// Mitsubishi GX Works2 project: PLC_GROUP6   PLC: FX3G

// global labels: Global1
VAR_GLOBAL
  startDay AT X007 : BOOL;
  lifeDay AT Y007 : BOOL;
  stayOn AT Y007 : BOOL;
  Dgima AT X001 : BOOL;
  AnalogInput1 AT D8280 : INT;
  beerType AT D1502 : REAL;
END_VAR
VAR_GLOBAL CONSTANT
  SHMARIMfor6_lagger : REAL := 150;
  LETETfor6_lagger : REAL := 12;
  KSHUTfor6_lagger : REAL := 60;
  SHMARIMfor6_pilzner : REAL := 120;
  LETETfor6_pilzner : REAL := 6;
  KSHUTfor6_pilzner : REAL := 54;
END_VAR
VAR_GLOBAL
  timerForCooking AT TC1 : BOOL;
END_VAR
VAR_GLOBAL CONSTANT
  secondsCooking : INT := 40;
END_VAR
VAR_GLOBAL
  EndCooking AT TS1 : BOOL;
  cooking AT Y001 : BOOL;
  stopCooking AT Y001 : BOOL;
  startTsisa AT X005 : BOOL;
  M0helper AT M0 : BOOL;
END_VAR
VAR_GLOBAL CONSTANT
  OnOf : INT := 5;
END_VAR
VAR_GLOBAL
  OnOfTsisa AT TC2 : BOOL;
  firstBulb AT TS2 : BOOL;
  first AT Y003 : BOOL;
  OnOfTsisa2 AT TC3 : BOOL;
  secondBulb AT TS3 : BOOL;
  second AT Y004 : BOOL;
  stopTsisa1 AT Y003 : BOOL;
  stopTsisa2 AT Y004 : BOOL;
  startAriza AT X002 : BOOL;
  arizat1Bottle AT X000 : BOOL;
  startMore5 AT Y002 : BOOL;
  countBottles AT CC1 : BOOL;
END_VAR
VAR_GLOBAL CONSTANT
  counterBottles : INT := 6;
END_VAR
VAR_GLOBAL
  finishCount AT CS1 : BOOL;
  endDay AT X011 : BOOL;
END_VAR
VAR_GLOBAL CONSTANT
  counterFirstBottle : INT := 1;
END_VAR
VAR_GLOBAL
  countFirstBottle AT CC0 : BOOL;
  startCount AT CS0 : BOOL;
  AddSixBeer AT Y002 : BOOL;
END_VAR
VAR_GLOBAL CONSTANT
  AddingSixBeer : REAL := 1.0;
END_VAR
VAR_GLOBAL
  validAmount AT M2 : BOOL;
  shmarim_Input AT D1100 : REAL;
  letet_Input AT D1200 : REAL;
  kshut_Input AT D1300 : REAL;
END_VAR
VAR_GLOBAL CONSTANT
  Min_shmarim : REAL := 120.0;
  Min_letet : REAL := 6.0;
  Min_kshut : REAL := 54.0;
END_VAR
VAR_GLOBAL
  shmarim_TOT AT D1102 : REAL;
  letet_TOT AT D1202 : REAL;
  kshut_TOT AT D1302 : REAL;
END_VAR
VAR_GLOBAL CONSTANT
  MinPIZ : REAL := 6.0;
END_VAR
VAR_GLOBAL
  checkValid AT M1 : BOOL;
  AmountSixBeer AT D1402 : REAL;
END_VAR
VAR_GLOBAL CONSTANT
  Normaliz : REAL := 404.5;
  MinLAG : REAL;
  MAXLAG : REAL := 5.0;
END_VAR
VAR_GLOBAL
  LAGChoose AT M3 : BOOL;
  PIZChoose AT M4 : BOOL;
  tsisaOfPIZ AT TC14 : BOOL;
  tsisaOfLAG AT TC13 : BOOL;
END_VAR
VAR_GLOBAL CONSTANT
  tsisaLAG : INT := 30;
  tsisaPIZ : INT := 40;
END_VAR
VAR_GLOBAL
  finishTSISAlag AT TS13 : BOOL;
  finishTSISApiz AT TS14 : BOOL;
  endOneIteration AT M10 : BOOL;
  theDayEnd AT M20 : BOOL;
END_VAR
VAR_GLOBAL CONSTANT
  constant_40 : REAL := 40;
END_VAR
VAR_GLOBAL
  Output_SixBeer AT D1404 : REAL;
  analogOutput AT D8282 : INT;
  checkMLAY AT M13 : BOOL;
END_VAR
VAR_GLOBAL CONSTANT
  bishul6LAG : REAL := 222;
END_VAR
VAR_GLOBAL
  bishul_TOT AT D1600 : REAL;
END_VAR
VAR_GLOBAL CONSTANT
  bishul6pilzner : REAL := 180;
END_VAR
VAR_GLOBAL
  tsisa_TOT AT D1602 : REAL;
  helpDayOn AT M22 : BOOL;
  endDayFINISH AT M11 : BOOL;
  MlayEndDay AT M12 : BOOL;
END_VAR

// task Task_01 (event TRUE, interval 0, priority 31): POU_01

PROGRAM POU_01
(* structured ladder/FBD written out as ST: instructions are called as NAME(EN, inputs, outputs); _pN, _eN, _tN stand for wires *)
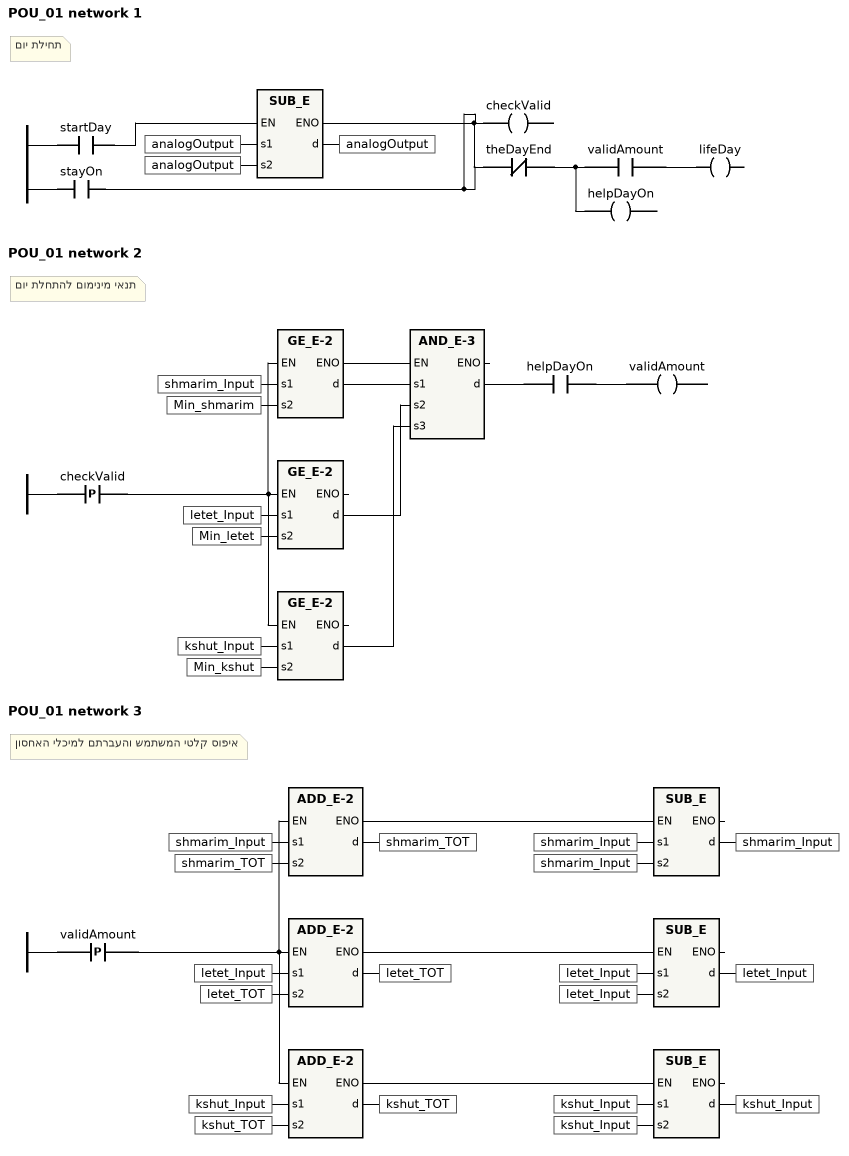
(* network 1 *)
(* תחילת יום *)
_e1 := SUB_E(startDay, analogOutput, analogOutput, analogOutput);
_p2 := _e1 OR stayOn;
checkValid := _p2;
_p3 := _p2 AND NOT theDayEnd;
lifeDay := _p3 AND validAmount;
helpDayOn := _p3;
(* network 2 *)
(* תנאי מינימום להתחלת יום *)
_p1 := LDP(TRUE, checkValid);
_e3 := GE_E(_p1, shmarim_Input, Min_shmarim, _t2);
GE_E(_p1, letet_Input, Min_letet, _t4);
GE_E(_p1, kshut_Input, Min_kshut, _t5);
AND_E(_e3, _t2, _t4, _t5, _t6);
validAmount := _t6 AND helpDayOn;
(* network 3 *)
(* איפוס קלטי המשתמש והעברתם למיכלי האחסון *)
_p1 := LDP(TRUE, validAmount);
_e2 := ADD_E(_p1, shmarim_Input, shmarim_TOT, shmarim_TOT);
SUB_E(_e2, shmarim_Input, shmarim_Input, shmarim_Input);
_e3 := ADD_E(_p1, letet_Input, letet_TOT, letet_TOT);
SUB_E(_e3, letet_Input, letet_Input, letet_Input);
_e4 := ADD_E(_p1, kshut_Input, kshut_TOT, kshut_TOT);
SUB_E(_e4, kshut_Input, kshut_Input, kshut_Input);
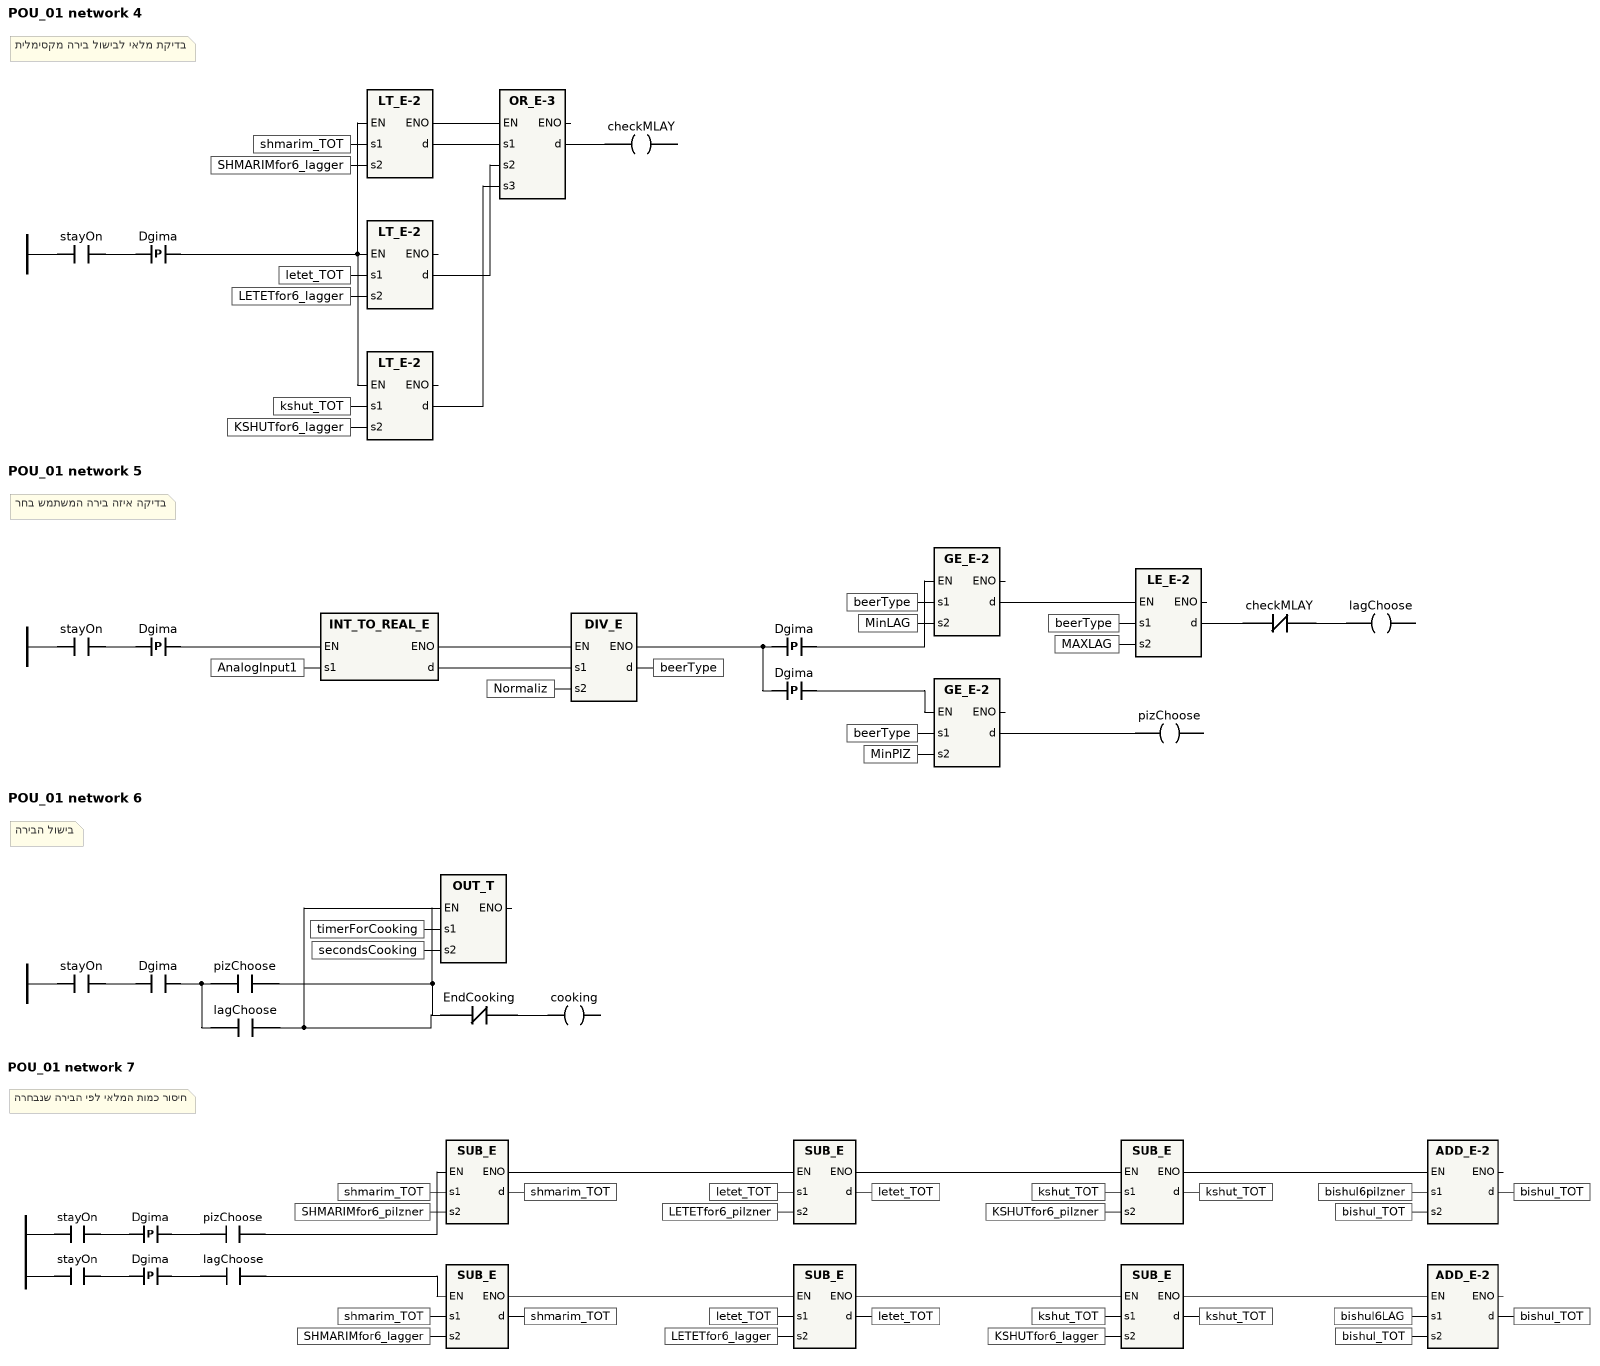
(* network 4 *)
(* בדיקת מלאי לבישול בירה מקסימלית *)
_p1 := stayOn AND LDP(TRUE, Dgima);
_e3 := LT_E(_p1, shmarim_TOT, SHMARIMfor6_lagger, _t2);
LT_E(_p1, letet_TOT, LETETfor6_lagger, _t4);
LT_E(_p1, kshut_TOT, KSHUTfor6_lagger, _t5);
OR_E(_e3, _t2, _t4, _t5, _t6);
checkMLAY := _t6;
(* network 5 *)
(* בדיקה איזה בירה המשתמש בחר *)
_e2 := INT_TO_REAL_E(stayOn AND LDP(TRUE, Dgima), AnalogInput1, _t1);
_e3 := DIV_E(_e2, _t1, Normaliz, beerType);
GE_E(_e3 AND LDP(TRUE, Dgima), beerType, MinLAG, _t4);
LE_E(_t4, beerType, MAXLAG, _t5);
lagChoose := _t5 AND NOT checkMLAY;
GE_E(_e3 AND LDP(TRUE, Dgima), beerType, MinPIZ, _t6);
pizChoose := _t6;
(* network 6 *)
(* בישול הבירה *)
_p1 := stayOn AND Dgima;
_p2 := (_p1 AND pizChoose) OR (_p1 AND lagChoose);
OUT_T(_p2, timerForCooking, secondsCooking);
cooking := _p2 AND NOT EndCooking;
(* network 7 *)
(* חיסור כמות המלאי לפי הבירה שנבחרה *)
_e1 := SUB_E(stayOn AND LDP(TRUE, Dgima) AND pizChoose, shmarim_TOT, SHMARIMfor6_pilzner, shmarim_TOT);
_e2 := SUB_E(_e1, letet_TOT, LETETfor6_pilzner, letet_TOT);
_e3 := SUB_E(_e2, kshut_TOT, KSHUTfor6_pilzner, kshut_TOT);
ADD_E(_e3, bishul6pilzner, bishul_TOT, bishul_TOT);
_e4 := SUB_E(stayOn AND LDP(TRUE, Dgima) AND lagChoose, shmarim_TOT, SHMARIMfor6_lagger, shmarim_TOT);
_e5 := SUB_E(_e4, letet_TOT, LETETfor6_lagger, letet_TOT);
_e6 := SUB_E(_e5, kshut_TOT, KSHUTfor6_lagger, kshut_TOT);
ADD_E(_e6, bishul6LAG, bishul_TOT, bishul_TOT);
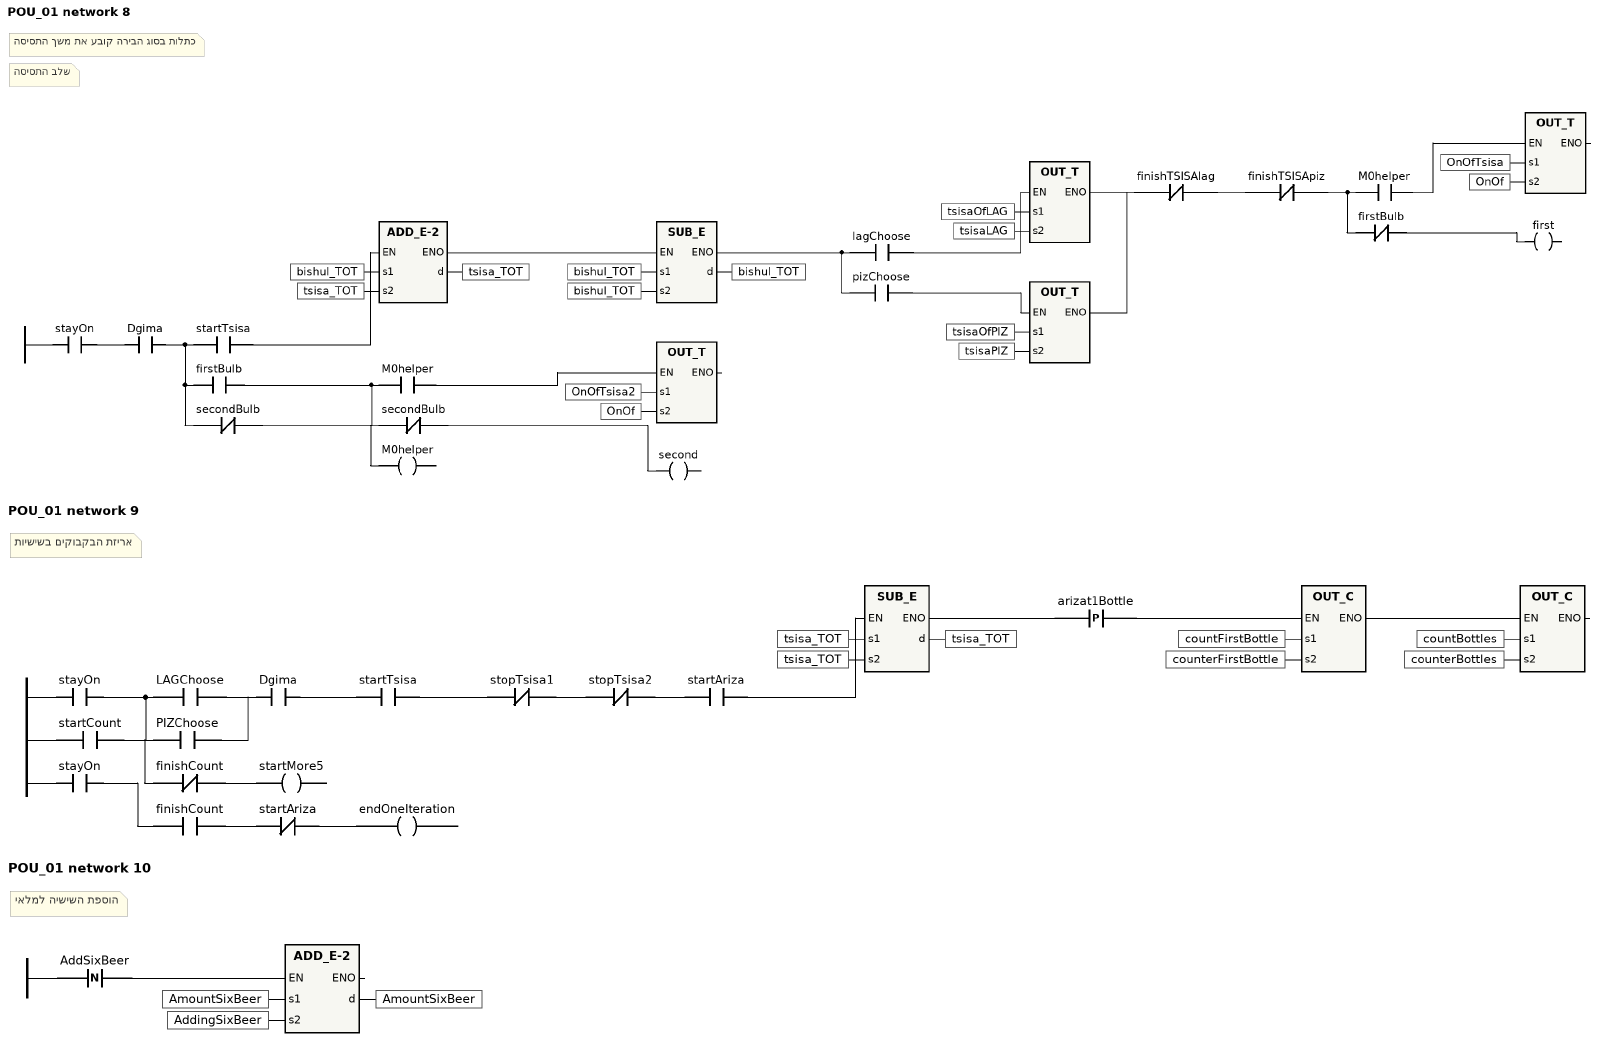
(* network 8 *)
(* כתלות בסוג הבירה קובע את משך התסיסה *)
(* שלב התסיסה *)
_p1 := stayOn AND Dgima;
_e2 := ADD_E(_p1 AND startTsisa, bishul_TOT, tsisa_TOT, tsisa_TOT);
_e3 := SUB_E(_e2, bishul_TOT, bishul_TOT, bishul_TOT);
_e4 := OUT_T(_e3 AND lagChoose, tsisaOfLAG, tsisaLAG);
_e5 := OUT_T(_e3 AND pizChoose, tsisaOfPIZ, tsisaPIZ);
_p6 := ((_e4 OR _e5) AND NOT finishTSISAlag) AND NOT finishTSISApiz;
OUT_T(_p6 AND M0helper, OnOfTsisa, OnOf);
first := _p6 AND NOT firstBulb;
_p7 := _p1 AND firstBulb;
OUT_T(_p7 AND M0helper, OnOfTsisa2, OnOf);
second := _p7 AND NOT secondBulb;
M0helper := _p1 AND NOT secondBulb;
(* network 9 *)
(* אריזת הבקבוקים בשישיות *)
_e1 := SUB_E(((((((stayOn AND LAGChoose) OR (stayOn AND PIZChoose)) AND Dgima) AND startTsisa) AND NOT stopTsisa1) AND NOT stopTsisa2) AND startAriza, tsisa_TOT, tsisa_TOT, tsisa_TOT);
_e2 := OUT_C(_e1 AND LDP(TRUE, arizat1Bottle), countFirstBottle, counterFirstBottle);
OUT_C(_e2, countBottles, counterBottles);
startMore5 := startCount AND NOT finishCount;
endOneIteration := stayOn AND finishCount AND NOT startAriza;
(* network 10 *)
(* הוספת השישיה למלאי *)
ADD_E(LDF(TRUE, AddSixBeer), AmountSixBeer, AddingSixBeer, AmountSixBeer);
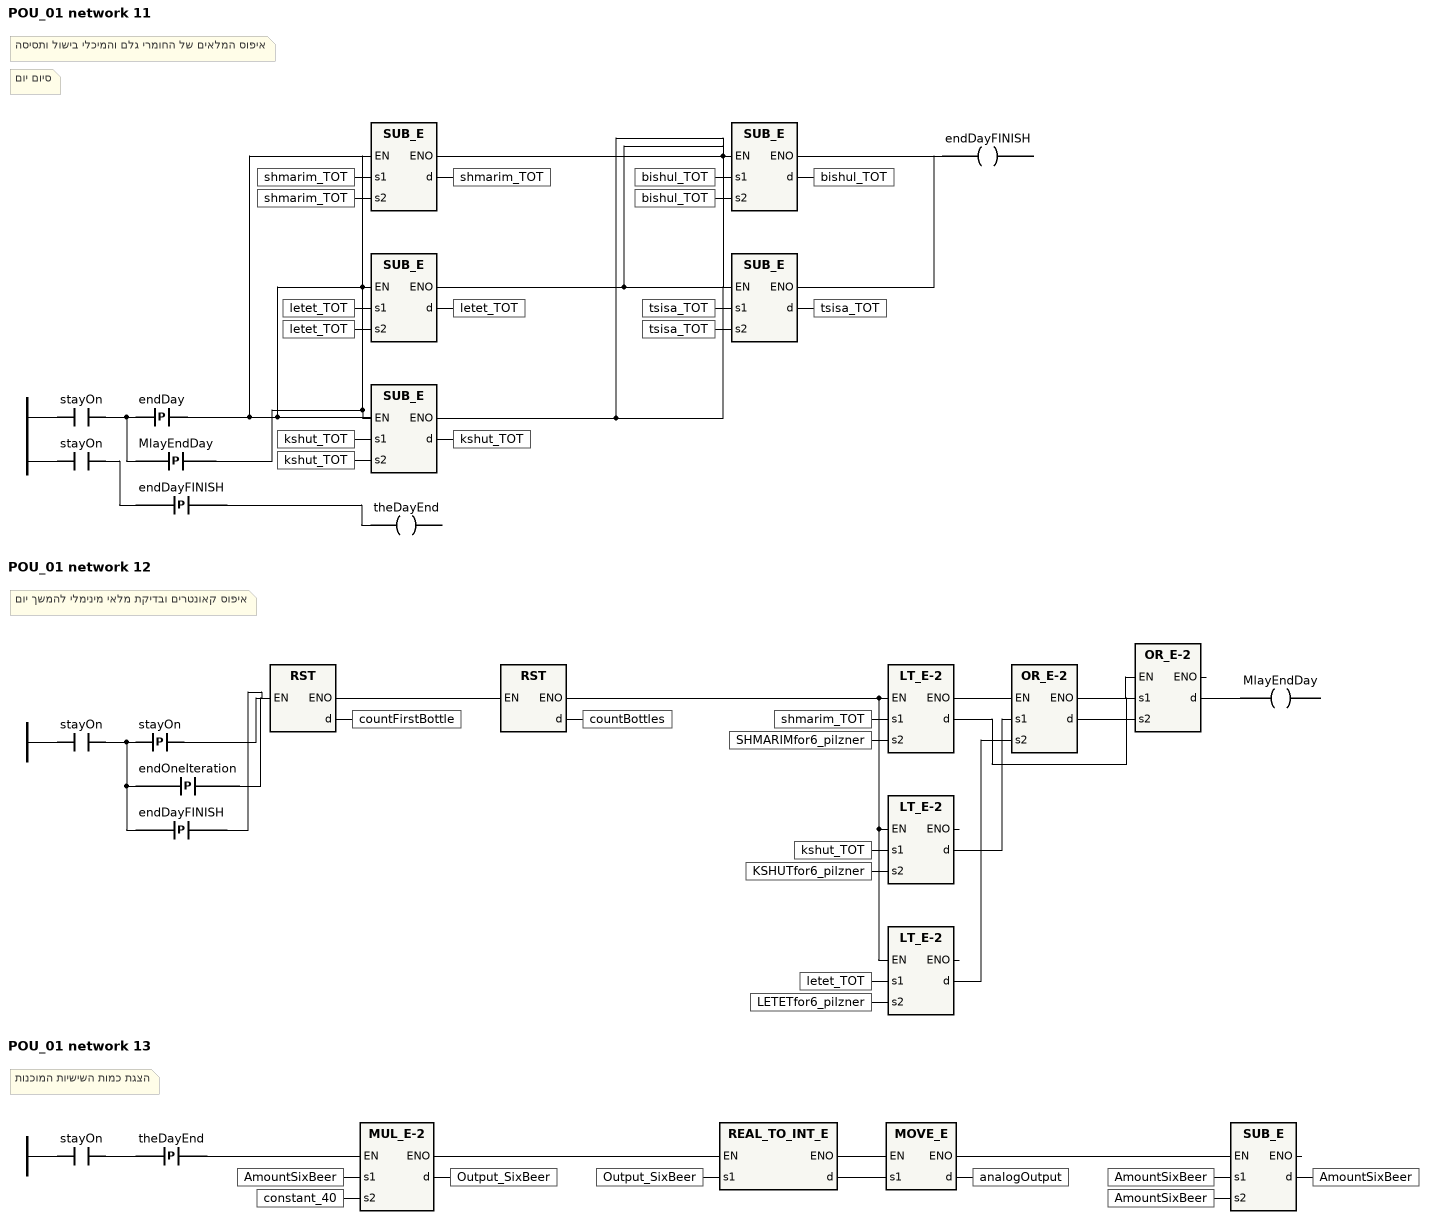
(* network 11 *)
(* איפוס המלאים של החומרי גלם והמיכלי בישול ותסיסה *)
(* סיום יום *)
_p1 := (stayOn AND LDP(TRUE, endDay)) OR (stayOn AND LDP(TRUE, MlayEndDay));
_e2 := SUB_E(_p1, shmarim_TOT, shmarim_TOT, shmarim_TOT);
_e3 := SUB_E(_p1, letet_TOT, letet_TOT, letet_TOT);
_e4 := SUB_E(_p1, kshut_TOT, kshut_TOT, kshut_TOT);
_p5 := _e2 OR _e3 OR _e4;
_e6 := SUB_E(_p5, bishul_TOT, bishul_TOT, bishul_TOT);
_e7 := SUB_E(_p5, tsisa_TOT, tsisa_TOT, tsisa_TOT);
endDayFINISH := _e6 OR _e7;
theDayEnd := stayOn AND LDP(TRUE, endDayFINISH);
(* network 12 *)
(* איפוס קאונטרים ובדיקת מלאי מינימלי להמשך יום *)
_e1 := RST((stayOn AND LDP(TRUE, stayOn)) OR (stayOn AND LDP(TRUE, endOneIteration)) OR (stayOn AND LDP(TRUE, endDayFINISH)), countFirstBottle);
_e2 := RST(_e1, countBottles);
_e4 := LT_E(_e2, shmarim_TOT, SHMARIMfor6_pilzner, _t3);
LT_E(_e2, kshut_TOT, KSHUTfor6_pilzner, _t5);
LT_E(_e2, letet_TOT, LETETfor6_pilzner, _t6);
_e8 := OR_E(_e4, _t5, _t6, _t7);
OR_E(_e8, _t3, _t7, _t9);
MlayEndDay := _t9;
(* network 13 *)
(* הצגת כמות השישיות המוכנות *)
_e1 := MUL_E(stayOn AND LDP(TRUE, theDayEnd), AmountSixBeer, constant_40, Output_SixBeer);
_e3 := REAL_TO_INT_E(_e1, Output_SixBeer, _t2);
_e4 := MOVE_E(_e3, _t2, analogOutput);
SUB_E(_e4, AmountSixBeer, AmountSixBeer, AmountSixBeer);
END_PROGRAM
